FUNCTION_BLOCK StartMotorsTask EXTENDS TcoUrRoboticsTask


IF Execute() THEN
    _blink(inOnTime := T#500MS, inOffTime := T#500MS);

    IF _progress = 0 THEN
        IF NOT __ISVALIDREF(inoControl) THEN
            _varInfo := __VARINFO(inoControl);
            Messenger.Programming(_sb.Clear().Append('<#Invalid reference: #>').Append(_varInfo.Symbol).ToString()).Pin();
        ELSIF NOT __ISVALIDREF(inoConfig) THEN
            _varInfo := __VARINFO(inoConfig);
            Messenger.Programming(_sb.Clear().Append('<#Invalid reference: #>').Append(_varInfo.Symbol).ToString()).Pin();
        ELSIF NOT __ISVALIDREF(inoStatus) THEN
            _varInfo := __VARINFO(inoStatus);
            Messenger.Programming(_sb.Clear().Append('<#Invalid reference: #>').Append(_varInfo.Symbol).ToString()).Pin();
        ELSE

            _progress := _progress + 1;

        END_IF

    END_IF

    IF _progress = 1 THEN
        THIS^.Messenger.OnCondition(_infoTimer.Q AND NOT inoStatus.State.Inputs.Safety.NO_IsNormalMode)
            .Warning(_sb.Clear().Append('<# Waiting to Normal Mode. #>').ToString());

        THIS^.Messenger.OnCondition(_infoTimer.Q AND NOT inoStatus.State.Inputs.Safety.RD_IsReducedMode)
            .Warning(_sb.Clear().Append('<# Waiting to Reduced Mode. #>').ToString());

        IF inoStatus.State.Inputs.Safety.NO_IsNormalMode OR inoStatus.State.Inputs.Safety.RD_IsReducedMode THEN
            _progress := _progress + 1;

        END_IF
    END_IF;

    IF _progress = 2 THEN
        Messenger.Warning('<#Robot has error Reset#>');

        IF NOT inoStatus.State.Inputs.Safety.FT_IsFault THEN
            _progress := _progress + 1;
        END_IF
    END_IF;

    IF _progress = 3 THEN
        Messenger.Debug('<#Robot Emergency Stop Reset#>');
        _varInfo := __VARINFO(inoStatus.State.Inputs.Safety.ES_IsEmergencyStopped);
        THIS^.Messenger.OnCondition(_infoTimer.Q AND NOT inoStatus.State.Inputs.Safety.ES_IsEmergencyStopped)
            .Warning(_sb.Clear().Append('<# Waiting for signal: #>').Append(_varInfo.Symbol).ToString());

        _varInfo := __VARINFO(inoStatus.State.Inputs.Safety.PS_IsProtectiveStopped);
        THIS^.Messenger.OnCondition(_infoTimer.Q AND NOT inoStatus.State.Inputs.Safety.PS_IsProtectiveStopped)
            .Warning(_sb.Clear().Append('<# Waiting for signal: #>').Append(_varInfo.Symbol).ToString());

        _varInfo := __VARINFO(inoStatus.State.Inputs.Safety.SS_IsSafeguardStopped);
        THIS^.Messenger.OnCondition(_infoTimer.Q AND NOT inoStatus.State.Inputs.Safety.SS_IsSafeguardStopped)
            .Warning(_sb.Clear().Append('<# Waiting for signal: #>').Append(_varInfo.Symbol).ToString());

        _varInfo := __VARINFO(inoStatus.State.Inputs.Safety.RC_IsRecoveryMode);
        THIS^.Messenger.OnCondition(_infoTimer.Q AND NOT inoStatus.State.Inputs.Safety.RC_IsRecoveryMode)
            .Warning(_sb.Clear().Append('<# Waiting for signal: #>').Append(_varInfo.Symbol).ToString());

        _varInfo := __VARINFO(inoStatus.State.Inputs.Safety.ST_IsStoppedDueSafety);
        THIS^.Messenger.OnCondition(_infoTimer.Q AND NOT inoStatus.State.Inputs.Safety.ES_IsEmergencyStopped)
            .Warning(_sb.Clear().Append('<# Waiting for signal: #>').Append(_varInfo.Symbol).ToString());

        _varInfo := __VARINFO(inoStatus.State.Inputs.Safety.VL_IsViolation);
        THIS^.Messenger.OnCondition(_infoTimer.Q AND NOT inoStatus.State.Inputs.Safety.VL_IsViolation)
            .Warning(_sb.Clear().Append('<# Waiting for signal: #>').Append(_varInfo.Symbol).ToString());

        //inoControl.ResetEmgStop := inoStatus.State.EmgStop AND _blink.outQ;
        IF NOT inoStatus.State.Inputs.Safety.ES_IsEmergencyStopped AND
            NOT inoStatus.State.Inputs.Safety.PS_IsProtectiveStopped AND
            NOT inoStatus.State.Inputs.Safety.SS_IsSafeguardStopped AND
            NOT inoStatus.State.Inputs.Safety.RC_IsRecoveryMode AND
            NOT inoStatus.State.Inputs.Safety.ST_IsStoppedDueSafety AND
            NOT inoStatus.State.Inputs.Safety.VL_IsViolation THEN
            //inoControl.ResetEmgStop:=FALSE;
            _progress := _progress + 1;
        END_IF
    END_IF;

    IF _progress = 4 THEN
        IF inoStatus.State.Inputs.Safety.FT_IsFault THEN
            _progress := 1;
        END_IF

        Messenger.Debug('<#Robot Power on#>');
        _varInfo := __VARINFO(inoStatus.State.Inputs.Robot.PW_IsPowerOn);
        THIS^.Messenger.OnCondition(_infoTimer.Q AND NOT inoStatus.State.Inputs.Robot.PW_IsPowerOn)
            .Warning(_sb.Clear().Append('<# Waiting for signal: #>').Append(_varInfo.Symbol).ToString());

        _varInfo := __VARINFO(inoStatus.State.Inputs.Safety.FT_IsFault);
        THIS^.Messenger.OnCondition(_infoTimer.Q AND NOT inoStatus.State.Inputs.Safety.FT_IsFault)
            .Warning(_sb.Clear().Append('<# Waiting for signal: #>').Append(_varInfo.Symbol).ToString());

        inoControl.MotorOn := _blink.outQ;

        IF inoStatus.State.Inputs.Robot.PW_IsPowerOn AND NOT inoStatus.State.Inputs.Safety.FT_IsFault AND
		    inoStatus.State.Inputs.Joints.JointMode[0] = 253 AND
            inoStatus.State.Inputs.Joints.JointMode[1] = 253 AND
            inoStatus.State.Inputs.Joints.JointMode[2] = 253 AND
            inoStatus.State.Inputs.Joints.JointMode[3] = 253 AND
            inoStatus.State.Inputs.Joints.JointMode[4] = 253 AND
            inoStatus.State.Inputs.Joints.JointMode[5] = 253 THEN
            inoControl.MotorOn := FALSE;
            _progress := _progress + 1;
        END_IF
    END_IF;


    DoneWhen(inoStatus.State.Inputs.Robot.PW_IsPowerOn AND
            NOT inoStatus.State.Inputs.Safety.FT_IsFault AND
            inoStatus.State.Inputs.Joints.JointMode[0] = 253 AND
            inoStatus.State.Inputs.Joints.JointMode[1] = 253 AND
            inoStatus.State.Inputs.Joints.JointMode[2] = 253 AND
            inoStatus.State.Inputs.Joints.JointMode[3] = 253 AND
            inoStatus.State.Inputs.Joints.JointMode[4] = 253 AND
            inoStatus.State.Inputs.Joints.JointMode[5] = 253);

    CallTimers(TRUE);

    THIS^.ThrowWhen(_errorTimer.Q);

END_IF

IF THIS^.Error AND NOT _errorMessage.Pinned THEN
    THIS^.Restore();
END_IF

(*~
	<docu>
		<summary>
			Executes when task is aborted.
		</summary>			
	</docu>	
~*)
METHOD PROTECTED OnAbort
IF  __ISVALIDREF(inoStatus) THEN   THIS^.inoStatus.ActionDescription := '<#Start motors  was aborted.#>'; END_IF;
END_METHOD

(*~
	<docu>
		<summary>
			Executes when task reaches the ```Done``` state .
		</summary>			
	</docu>	
~*)
METHOD PROTECTED OnDone
IF  __ISVALIDREF(inoStatus) THEN   THIS^.inoStatus.ActionDescription := '<#Start motors  finished successfully.#>'; END_IF;
_progress:=0;
END_METHOD

METHOD PROTECTED OnError
VAR
	description: STRING;
END_VAR
description := '<#Start motors finished with error.#>'; 
IF  __ISVALIDREF(inoStatus) THEN   THIS^.inoStatus.ActionDescription := description; END_IF;
THIS^._errorMessage.Error(_sb.Clear().Append(description).Append(' To restore acknowledge this alarm.').ToString()).Pin();
END_METHOD

METHOD PROTECTED OnStart
IF  __ISVALIDREF(inoStatus) THEN  THIS^.inoStatus.ActionDescription := '<#Start motors started.#>'; END_IF; 
CallTimers(FALSE);
END_METHOD

(*~
	<docu>
		<summary>
			Restores this instance to the Ready state. Can be called explicitly or from within one of the restore mechanisms.
			<para>
				See also <see cref="PlcDocu.TcoCore.TcoTask.AutoRestorable()"/>
			</para>
		</summary>			
	</docu>	
~*)
METHOD Restore : ITcoRestorable
SUPER^.Restore();
END_METHOD

END_FUNCTION_BLOCK

(* stored: Version 1.1.0.1, ProductVersion 3.1.4024.12
   POU StartMotorsTask: Id {5a26caf7-d182-024b-3225-4bd4a5c39f1d}, SpecialFunc None
   Method OnAbort: Id {232ebecc-cbbc-0a34-338c-20e2cd172bea}
   Method OnDone: Id {fcacdbbb-0470-097b-0337-5843fe8a4a29}
   Method OnError: Id {8a72d4a8-165e-0e81-237a-36e3ffb97947}
   Method OnStart: Id {824a9fb4-6b86-0ff1-3d9b-f6c0df651a44}
   Method Restore: Id {13baab1c-4a82-0472-260c-87ca0a14773b} *)
